FUNCTION_BLOCK fbIfElse
VAR_INPUT
	BVal		:BOOL;
	IFVal		:REAL;
	ELSEVal		:REAL;
END_VAR
VAR_OUTPUT
	OUT			:REAL;
END_VAR
VAR
END_VAR

IF BVal THEN
	OUT := IFVal;
ELSE
	OUT := ELSEVal;
END_IF

END_FUNCTION_BLOCK

(* stored: Version 1.1.0.1, ProductVersion 3.1.4022.6
   POU fbIfElse: Id {8994fbc7-7e06-44d7-b2cc-1f65de126893}, SpecialFunc None *)
